INTERFACE I_SuperBohrmachine

METHOD Bohren : HRESULT
END_METHOD

METHOD Start : HRESULT
VAR_INPUT
	config: REFERENCE TO ST_Config;
END_VAR
END_METHOD

METHOD Stop : HRESULT
VAR_INPUT
END_VAR
END_METHOD

END_INTERFACE

(* stored: Version 1.1.0.1, ProductVersion 3.1.4024.3
   Itf I_SuperBohrmachine: Id {7e529ac0-6fa6-4842-8bba-6c0ea8e5d5f9}
   Method Bohren: Id {a936cd81-6d0e-45c8-9ffa-f169333734b4}
   Method Start: Id {a54a25fa-479d-4f3c-a002-2897e85c7eaf}
   Method Stop: Id {5142dc78-5cae-4990-ad95-dd8064b0a39c} *)
